FUNCTION Convert_BOOL_TO_REAL : BOOL
VAR_INPUT
	in : BOOL;
	out : REFERENCE TO REAL;
END_VAR
VAR
	converted : REAL;
END_VAR

converted := BOOL_TO_REAL(in);

IF (REAL_TO_BOOL(converted) <> in) THEN
	RETURN;
END_IF

out := converted;
Convert_BOOL_TO_REAL := TRUE;

END_FUNCTION

(* stored: Version 1.1.0.1, ProductVersion 3.1.4024.12
   POU Convert_BOOL_TO_REAL: Id {6aebb5f9-4071-4ecb-a38a-5d2bec8518f1}, SpecialFunc None *)
